TYPE T_CASE_Barcode : T_MaxString;
END_TYPE

(* stored: Version 1.1.0.1
   DUT T_CASE_Barcode: Id {a823e532-93bb-46e4-a5a1-473471c3594f} *)
